PROGRAM MAIN
VAR
	Ladder : POU_MainFunc;
	Motor: POU_NCPowerOn;
	ReadXAxisStatus:MC_ReadStatus;
	poweraxis: MC_PowerStepper;
	resetaxis: MC_Reset;
	stopaxis: MC_Stop;
	MoveVelocity: MC_MoveVelocity;
	direction: MC_Direction;
	SetVel: MC_MoveAbsolute;
	
	
END_VAR


	
	
Ladder();
motor();

END_PROGRAM

(* stored: Version 1.1.0.1, ProductVersion 3.1.4024.2
   POU MAIN: Id {eaaaa866-ff64-4f1f-a8a1-5273cc9f3e0d}, SpecialFunc None *)
